Universal Robots PolyScope program: iniciales1-nombres.urp

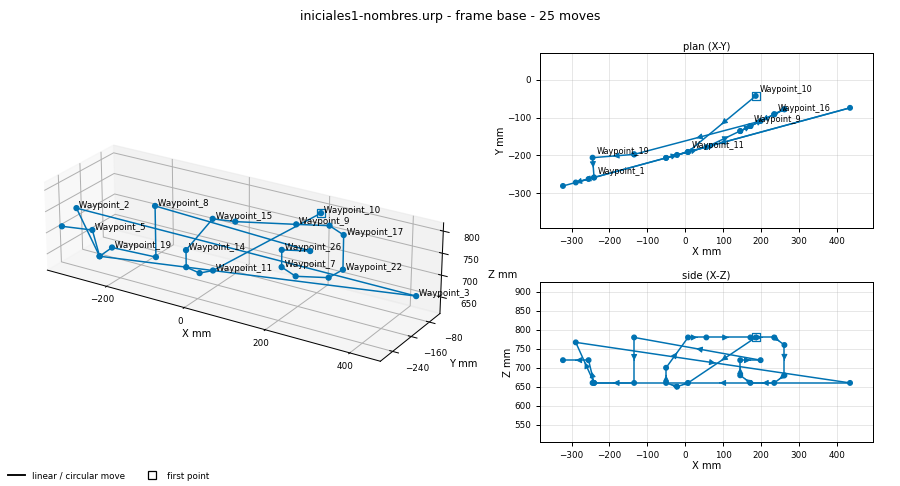
[picture p0: tool path of iniciales1-nombres.urp in frame base, 25 of 25 moves have a stored position in this frame; points joined in program order, loops and branches not executed]
Program iniciales1-nombres (installation=default directory=/ursim/programs createdIn=3.15.8.106339 lastSavedIn=3.15.8.106339 robotSerialNumber=2018359999)
Calibrated DH parameters: a=[0, -0.425, -0.39225, 0, 0, 0]; d=[0.089159, 0, 0, 0.10915, 0.09465, 0.0823]; alpha=[1.570796, 0, 0, 1.570796, -1.570796, 0]; deltaTheta=[0, 0, 0, 0, 0, 0]
Robot Program (runOnlyOnce=false)
  Popup Message (haltProgram=true message=se va a realizar la letra J inputType=Text)
  MoveL speed 250 mm/s, acceleration 1200 mm/s^2 (useActiveTCP=true) feature=Base
    Waypoint Waypoint_10: TCP in base x=186 y=-43 z=780 mm, rx=-0.0012 ry=3.1163 rz=0.0389 rad; joints [21.432, -76.168, -38.187, -153.785, 90.807, 111.4] deg
    Wait Sleep waitTime=0.5
    Waypoint Waypoint_11: TCP in base x=7.358 y=-190.764 z=660 mm, rx=-0.0012 ry=3.1163 rz=0.0389 rad; joints [-53.964, -60.773, -73.111, -136.428, 92.003, 35.985] deg
    Wait Sleep waitTime=0.5
    Waypoint Waypoint_12: TCP in base x=-21.589 y=-198.643 z=650 mm, rx=-0.0012 ry=3.1163 rz=0.0389 rad; joints [-64.029, -60.929, -75.023, -134.706, 91.917, 25.915] deg
    Wait Sleep waitTime=0.5
    Waypoint Waypoint_13: TCP in base x=-50.535 y=-206.522 z=660 mm, rx=-0.0012 ry=3.1163 rz=0.0389 rad; joints [-73.661, -63.5, -72.12, -135.348, 91.78, 16.279] deg
    Wait Sleep waitTime=0.5
    Waypoint Waypoint_14: TCP in base x=-50.535 y=-206.522 z=700 mm, rx=-0.0012 ry=3.1163 rz=0.0389 rad; joints [-73.661, -67.802, -62.037, -141.13, 91.78, 16.279] deg
    Wait Sleep waitTime=0.5
    Waypoint Waypoint_15: TCP in base x=7.358 y=-190.764 z=780 mm, rx=-0.0012 ry=3.1163 rz=0.0389 rad; joints [-53.964, -77.28, -36.468, -156.564, 92.003, 35.985] deg
    Wait Sleep waitTime=0.5
    Waypoint Waypoint_25: TCP in base x=55.719 y=-178.056 z=780 mm, rx=-0.0392 ry=2.2037 rz=-2.2037 rad; joints [32.733, -48.252, -86.387, -45.361, -30.709, -0.012] deg
  Popup Message (haltProgram=true message=se va a realizar la letra G inputType=Text)
  MoveL speed 250 mm/s, acceleration 1200 mm/s^2 (useActiveTCP=true) feature=Base
    Waypoint Waypoint_9: TCP in base x=171.977 y=-122.555 z=780 mm, rx=-0.0012 ry=3.1163 rz=0.0389 rad; joints [-5.056, -78.729, -36.74, -153.226, 91.551, 84.917] deg
    Wait Sleep waitTime=0.5
    Waypoint Waypoint_16: TCP in base x=234.752 y=-91.583 z=780 mm, rx=0 ry=2.2214 rz=-2.2214 rad; joints [150.052, -108.321, 78.891, -150.57, -150.052, 0] deg
    Wait Sleep waitTime=0.5
    Waypoint Waypoint_17: TCP in base x=261.656 y=-78.309 z=760 mm, rx=-0.0392 ry=2.2037 rz=-2.2037 rad; joints [25.82, -118.15, 23.159, 94.991, 23.796, -180.012] deg
    Wait Sleep waitTime=0.5
    Waypoint Waypoint_22: TCP in base x=261.656 y=-78.309 z=680 mm, rx=-0.0392 ry=2.2037 rz=-2.2037 rad; joints [155.925, -19.368, -95.719, -64.913, -153.901, -0.012] deg
    Wait Sleep waitTime=0.5
    Waypoint Waypoint_23: TCP in base x=234.752 y=-91.583 z=660 mm, rx=-0.0392 ry=2.2037 rz=-2.2037 rad; joints [25.755, -65.378, -101.382, -13.239, -23.731, -0.012] deg
    Wait Sleep waitTime=0.5
    Waypoint Waypoint_24: TCP in base x=171.977 y=-122.555 z=660 mm, rx=-0.0392 ry=2.2037 rz=-2.2037 rad; joints [25.493, -56.098, -105.559, -18.343, -23.469, -0.012] deg
    Wait Sleep waitTime=0.5
    Waypoint Waypoint_7: TCP in base x=145.074 y=-135.829 z=680 mm, rx=-0.0392 ry=2.2037 rz=-2.2037 rad; joints [25.274, -53.241, -103.372, -23.387, -23.25, -0.012] deg
    Wait Sleep waitTime=0.5
    Waypoint Waypoint_26: TCP in base x=145.074 y=-135.829 z=720 mm, rx=-0.0392 ry=2.2037 rz=-2.2037 rad; joints [25.274, -55.622, -96.167, -28.211, -23.25, -0.012] deg
    Wait Sleep waitTime=0.5
    Waypoint Waypoint_27: TCP in base x=198.881 y=-109.281 z=720 mm, rx=-0.0392 ry=2.2037 rz=-2.2037 rad; joints [138.66, -117.16, 93.398, -156.238, -136.636, -0.012] deg
  Popup Message (haltProgram=true message=se va a realizar la letra L inputType=Text)
  MoveL speed 250 mm/s, acceleration 1200 mm/s^2 (useActiveTCP=true) feature=Base
    Waypoint Waypoint_8: TCP in base x=-134.857 y=-197.255 z=780 mm, rx=-0.0392 ry=2.2037 rz=-2.2037 rad; joints [2.394, -37.142, -82.893, -59.965, -0.371, -0.012] deg
    Wait Sleep waitTime=0.5
    Waypoint Waypoint_18: TCP in base x=-134.857 y=-197.255 z=660 mm, rx=-0.0392 ry=2.2037 rz=-2.2037 rad; joints [2.394, -23.745, -105.203, -51.052, -0.371, -0.012] deg
    Wait Sleep waitTime=0.5
    Waypoint Waypoint_19: TCP in base x=-244.515 y=-205.934 z=660 mm, rx=-0.0392 ry=2.2037 rz=-2.2037 rad; joints [-130.199, -71.988, -97.432, -10.58, 132.223, -0.012] deg
  Popup Message (haltProgram=true message=se va a realizar la letra J inputType=Text)
  MoveL speed 250 mm/s, acceleration 1200 mm/s^2 (useActiveTCP=true) feature=Base
    Waypoint Waypoint_1: TCP in base x=-240.62 y=-258.259 z=660 mm, rx=-0.0012 ry=3.1163 rz=0.0389 rad; joints [-115.132, -80.716, -62.148, -129.041, 90.692, -25.189] deg
    Wait Sleep waitTime=0.5
    Waypoint Waypoint_2: TCP in base x=-288.865 y=-271.391 z=767 mm, rx=-0.0012 ry=3.1163 rz=0.0389 rad; joints [-120.909, -108.219, -5.309, -158.437, 90.497, -30.962] deg
    Wait Sleep waitTime=0.5
    Waypoint Waypoint_3: TCP in base x=434.808 y=-74.419 z=660 mm, rx=-0.0012 ry=3.1163 rz=0.0389 rad; joints [4.36, -91.379, -53.499, -123.581, 91.317, 94.333] deg
    Wait Sleep waitTime=0.5
    Waypoint Waypoint_4: TCP in base x=-240.62 y=-258.259 z=660 mm, rx=-0.0012 ry=3.1163 rz=0.0389 rad; joints [-115.132, -80.716, -62.148, -129.041, 90.692, -25.189] deg
    Wait Sleep waitTime=0.5
    Waypoint Waypoint_5: TCP in base x=-255.094 y=-262.199 z=720 mm, rx=-0.0012 ry=3.1163 rz=0.0389 rad; joints [-117.001, -89.315, -42.728, -139.884, 90.63, -27.057] deg
    Wait Sleep waitTime=0.5
    Waypoint Waypoint_6: TCP in base x=-322.636 y=-280.583 z=720 mm, rx=-0.0012 ry=3.1163 rz=0.0389 rad; joints [-124.274, -98.777, -32.152, -141.062, 90.381, -34.325] deg
